PROGRAM LightsTest
VAR
	fbLightTestOn_TRIG: R_TRIG;
	fbLightTestOff_TRIG: F_TRIG;
 	xLightTest:BOOL;
END_VAR

LightsTest();

ACTION LightsTest:
fbLightTestOn_TRIG(CLK:=xLightTest , Q=> );
fbLightTestOff_TRIG(CLK:=xLightTest , Q=> );
IF fbLightTestOn_TRIG.Q THEN
	QxStartButtonLamp:=TRUE	;//	启动按钮指示灯
	QxStopButtonLamp:=TRUE		;//	停止按钮指示灯
  QxResetButtonLamp:=TRUE		;//	复位按钮指示灯
  QxInitButtonLamp:=TRUE		;//	初始化按钮指示灯
	QxMachineLamp1Control:=TRUE;	;//	日光灯1控制
  QxMachineLamp2Control:=TRUE;	;//	日光灯2控制
	QxRedLamp	:=TRUE;//	三色灯-红灯
	QxYellowLamp:=TRUE	;//	三色灯-黄灯
	QxGreenLamp:=TRUE	;//	三色灯-绿灯
	QxCameraLight1Trigger:=TRUE	;//	相机光源触发通道1
	QxCameraLight2Trigger:=TRUE	;//	相机光源触发通道2
	QxCameraLight3Trigger:=TRUE	;//	相机光源触发通道3
	QxCameraLight4Trigger:=TRUE	;//	相机光源触发通道4
	
	QxRedLamp_1:=TRUE	;//	三色灯-红灯
	QxYellowLamp_1:=TRUE	;//	三色灯-黄灯
  QxGreenLamp_1:=TRUE	;//	三色灯-绿灯
	QxMachineLamp3Contorl:=TRUE	;//	日光灯控制
ELSIF fbLightTestOff_TRIG.Q THEN
	QxStartButtonLamp:=FALSE	;//	启动按钮指示灯
	QxStopButtonLamp:=FALSE		;//	停止按钮指示灯
  QxResetButtonLamp:=FALSE		;//	复位按钮指示灯
  QxInitButtonLamp:=FALSE		;//	初始化按钮指示灯
	QxMachineLamp1Control:=FALSE;	;//	日光灯1控制
  QxMachineLamp2Control:=FALSE;	;//	日光灯2控制
	QxRedLamp	:=FALSE;//	三色灯-红灯
	QxYellowLamp:=FALSE	;//	三色灯-黄灯
	QxGreenLamp:=FALSE	;//	三色灯-绿灯
	QxCameraLight1Trigger:=FALSE	;//	相机光源触发通道1
	QxCameraLight2Trigger:=FALSE	;//	相机光源触发通道2
	QxCameraLight3Trigger:=FALSE	;//	相机光源触发通道3
	QxCameraLight4Trigger:=FALSE	;//	相机光源触发通道4
	
	QxRedLamp_1:=FALSE	;//	三色灯-红灯
	QxYellowLamp_1:=FALSE	;//	三色灯-黄灯
  QxGreenLamp_1:=FALSE	;//	三色灯-绿灯
	QxMachineLamp3Contorl:=FALSE	;//	日光灯控制
END_IF
END_ACTION

END_PROGRAM

(* stored: Version 1.1.0.1, ProductVersion 3.1.4024.9
   POU LightsTest: Id {1146d2cb-f55d-4151-aa2a-43669887c966}, SpecialFunc None
   Action LightsTest: Id {436fc6ec-8d98-4c22-8d21-a7095f64a587} *)
